# EPICS autosave request: iocBoot/iocMKS946/mks946_settings.req
$(P)$(MFC):setscalefactor
$(P)$(MFC):setscalerange
$(P)$(MFC):setpoint
$(P)$(MFC):setmode
